# EPICS autosave request: ipApp/Db/PTC10_aio_chan_settings.req
$(P)$(T):$(C):ioType
$(P)$(T):$(C):setPoint
$(P)$(T):$(C):rampRate
$(P)$(T):$(C):pid:P
$(P)$(T):$(C):pid:I
$(P)$(T):$(C):pid:D
$(P)$(T):$(C):pid:input
$(P)$(T):$(C):output
$(P)$(T):$(C):output_RBV.SCAN
$(P)$(T):$(C):rampTemp_RBV.SCAN
$(P)$(T):$(C):tune:lag
$(P)$(T):$(C):tune:step
$(P)$(T):$(C):tune:type
$(P)$(T):$(C):poll.SCAN
